// TIA Portal V15.1 export
// export: Created 2020-06-12T07:35:40.4599609Z, ExportSetting None, DisplayName Totally Integrated Automation Portal, DisplayVersion V15.1, DisplayName TIA Portal Openness, DisplayVersion V15.1, DisplayName STEP 7 Professional, DisplayVersion V15.1, DisplayName STEP 7 Safety, DisplayVersion V15.1, DisplayName WinCC Advanced, DisplayVersion V15.1
DATA_BLOCK "F_data"   // DB609, F_DB
{ S7_Optimized_Access := 'TRUE' }
   VAR
      emer_undel_on { ExternalAccessible := 'False'; ExternalVisible := 'False'; ExternalWritable := 'False'} : Bool := TRUE;   // Emergency line Undelayed ok
      emer_del_on { ExternalAccessible := 'False'; ExternalVisible := 'False'; ExternalWritable := 'False'} : Bool := TRUE;   // Emergency line Delayed ok
      sd_undel_on { ExternalAccessible := 'False'; ExternalVisible := 'False'; ExternalWritable := 'False'} : Bool := TRUE;   // Emergency & SDoors line Undelayed ok
      sd_del_on { ExternalAccessible := 'False'; ExternalVisible := 'False'; ExternalWritable := 'False'} : Bool := TRUE;   // Emergency & SDoors line Delayed ok
      mcb_rel_undel { ExternalAccessible := 'False'; ExternalVisible := 'False'; ExternalWritable := 'False'} : Bool := FALSE;   // MCB release undelayed ok
      mcb_rel_del { ExternalAccessible := 'False'; ExternalVisible := 'False'; ExternalWritable := 'False'} : Bool := FALSE;   // MCB release delayed ok
      trafo_sup_undel { ExternalAccessible := 'False'; ExternalVisible := 'False'; ExternalWritable := 'False'} : Bool := TRUE;   // Trafo supply on (undelayed)
      trafo_rel { ExternalAccessible := 'False'; ExternalVisible := 'False'; ExternalWritable := 'False'} : Bool := TRUE;   // Trafo release (delayed)
      ES1YM01_emer_undel_on { ExternalAccessible := 'False'; ExternalVisible := 'False'; ExternalWritable := 'False'} : Bool := TRUE;   // Emergency line Undelayed out
      ES1YM01_emer_undel_err { ExternalAccessible := 'False'; ExternalVisible := 'False'; ExternalWritable := 'False'} : Bool := FALSE;   // Emergency line Undelayed error
      ES1YM01_emer_del_on { ExternalAccessible := 'False'; ExternalVisible := 'False'; ExternalWritable := 'False'} : Bool := TRUE;   // Emergency line Delayed out
      ES1YM01_emer_del_err { ExternalAccessible := 'False'; ExternalVisible := 'False'; ExternalWritable := 'False'} : Bool := FALSE;   // Emergency line Delayed error
      ES1LA1_M01_err { ExternalAccessible := 'False'; ExternalVisible := 'False'; ExternalWritable := 'False'} : Bool := FALSE;   // Screw Conveyer release Error
      ES1LE1_EV02_rel_on { ExternalAccessible := 'False'; ExternalVisible := 'False'; ExternalWritable := 'False'} : Bool := TRUE;   // Spindle Break Release on
      ES1LE1_EV02_rel_err { ExternalAccessible := 'False'; ExternalVisible := 'False'; ExternalWritable := 'False'} : Bool := FALSE;   // Spindle Break Release error
      ES1LE1_M01_rel_on { ExternalAccessible := 'False'; ExternalVisible := 'False'; ExternalWritable := 'False'} : Bool := TRUE;   // Electrode Carriage Safe Release on
      ES1LE1_M01_rel_err { ExternalAccessible := 'False'; ExternalVisible := 'False'; ExternalWritable := 'False'} : Bool := FALSE;   // Electrode Carriage Safe Release error
      ES1LE2_M01_rel_err { ExternalAccessible := 'False'; ExternalVisible := 'False'; ExternalWritable := 'False'} : Bool := FALSE;   // X-Drive Safe Release error
      ES1LE2_M02_rel_err { ExternalAccessible := 'False'; ExternalVisible := 'False'; ExternalWritable := 'False'} : Bool := FALSE;   // Y-Drive Safe Release error
      ES1LE3_M01_rel_on { ExternalAccessible := 'False'; ExternalVisible := 'False'; ExternalWritable := 'False'} : Bool := TRUE;   // Protective Gas Hood Safe Release on
      ES1LE3_M01_rel_err { ExternalAccessible := 'False'; ExternalVisible := 'False'; ExternalWritable := 'False'} : Bool := FALSE;   // Protective Gas Hood Safe Release error
      ES1LE4_EV01_rel_on { ExternalAccessible := 'False'; ExternalVisible := 'False'; ExternalWritable := 'False'} : Bool := TRUE;   // Pneumatic Valve Power Ram Safe Release on
      ES1LE4_EV01_rel_err { ExternalAccessible := 'False'; ExternalVisible := 'False'; ExternalWritable := 'False'} : Bool := FALSE;   // Pneumatic Valve Power Ram Safe Release error
      ES1LE4_EV02_rel_on { ExternalAccessible := 'False'; ExternalVisible := 'False'; ExternalWritable := 'False'} : Bool := TRUE;   // Pneumatic Valve Current Pipes Cylinders Safe Release on
      ES1LE4_EV02_rel_err { ExternalAccessible := 'False'; ExternalVisible := 'False'; ExternalWritable := 'False'} : Bool := FALSE;   // Pneumatic Valve Current Pipes Cylinders Safe Release error
      ES1LE4_M01_rel_on { ExternalAccessible := 'False'; ExternalVisible := 'False'; ExternalWritable := 'False'} : Bool := TRUE;   // Portal Swiveling Safe Release on
      ES1LE4_M01_rel_err { ExternalAccessible := 'False'; ExternalVisible := 'False'; ExternalWritable := 'False'} : Bool := FALSE;   // Portal Swiveling Safe Release error
      ES1LM1_EV01_rel_on { ExternalAccessible := 'False'; ExternalVisible := 'False'; ExternalWritable := 'False'} : Bool := TRUE;   // Pneumatic Valve Baseplate Clamp MS1 Cylinders Safe Release on
      ES1LM1_EV01_rel_err { ExternalAccessible := 'False'; ExternalVisible := 'False'; ExternalWritable := 'False'} : Bool := FALSE;   // Pneumatic Valve Baseplate Clamp MS1 Cylinders Safe Release error
      ES1LM2_EV01_rel_on { ExternalAccessible := 'False'; ExternalVisible := 'False'; ExternalWritable := 'False'} : Bool := TRUE;   // Pneumatic Valve Baseplate Clamp MS2 Cylinders Safe Release on
      ES1LM2_EV01_rel_err { ExternalAccessible := 'False'; ExternalVisible := 'False'; ExternalWritable := 'False'} : Bool := FALSE;   // Pneumatic Valve Baseplate Clamp MS2 Cylinders Safe Release error
      ES1LS1_XS01_rel_on { ExternalAccessible := 'False'; ExternalVisible := 'False'; ExternalWritable := 'False'} : Bool := FALSE;   // MCB Safety Release on
      ES1LS1_XS01_rel_err { ExternalAccessible := 'False'; ExternalVisible := 'False'; ExternalWritable := 'False'} : Bool := FALSE;   // MCB Safety Release error
      ES1LE1_M01_STO { ExternalAccessible := 'False'; ExternalVisible := 'False'; ExternalWritable := 'False'} : Bool := TRUE;   // Electrode Carriage Safe Torque off Ok
      ES1LE1_M01_STO_err { ExternalAccessible := 'False'; ExternalVisible := 'False'; ExternalWritable := 'False'} : Bool := FALSE;   // Electrode Carriage Safe Torque off error
      ES1LE3_M01_STO { ExternalAccessible := 'False'; ExternalVisible := 'False'; ExternalWritable := 'False'} : Bool := TRUE;   // Protective Gas Hood Safe Torque off Ok
      ES1LE3_M01_STO_err { ExternalAccessible := 'False'; ExternalVisible := 'False'; ExternalWritable := 'False'} : Bool := FALSE;   // Protective Gas Hood Safe Torque off error
      ES1LE4_M01_STO { ExternalAccessible := 'False'; ExternalVisible := 'False'; ExternalWritable := 'False'} : Bool := TRUE;   // Portal Swiveling Safe Torque off Ok
      ES1LE4_M01_STO_err { ExternalAccessible := 'False'; ExternalVisible := 'False'; ExternalWritable := 'False'} : Bool := FALSE;   // Portal Swiveling Safe Torque off error
   END_VAR
BEGIN
END_DATA_BLOCK
